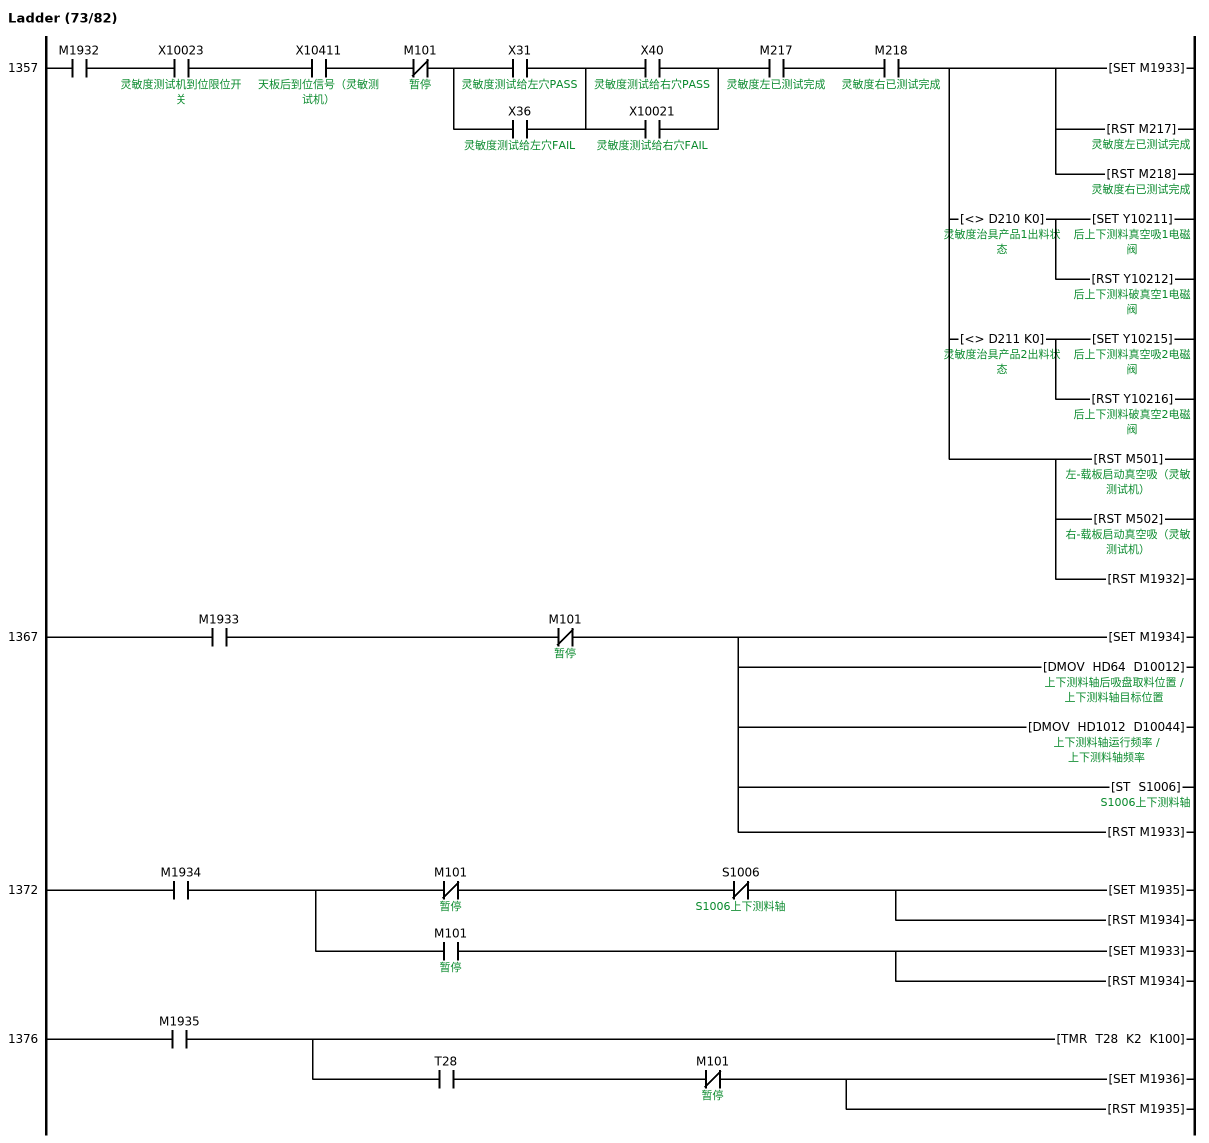
[picture p72: Ladder rows 1357-1376]
LD     M1932
AND    X10023	; 灵敏度测试机到位限位开关
AND    X10411	; 天板后到位信号（灵敏测试机）
ANI    M101	; 暂停
LD     X31	; 灵敏度测试给左穴PASS
OR     X36	; 灵敏度测试给左穴FAIL
ANB
LD     X40	; 灵敏度测试给右穴PASS
OR     X10021	; 灵敏度测试给右穴FAIL
ANB
AND    M217	; 灵敏度左已测试完成
AND    M218	; 灵敏度右已测试完成
SET    M1933
RST    M217	; 灵敏度左已测试完成
RST    M218	; 灵敏度右已测试完成
MPS
AND<>  D210 K0	; 灵敏度治具产品1出料状态
SET    Y10211	; 后上下测料真空吸1电磁阀
RST    Y10212	; 后上下测料破真空1电磁阀
MRD
AND<>  D211 K0	; 灵敏度治具产品2出料状态
SET    Y10215	; 后上下测料真空吸2电磁阀
RST    Y10216	; 后上下测料破真空2电磁阀
MPP
RST    M501	; 左-载板启动真空吸（灵敏测试机）
RST    M502	; 右-载板启动真空吸（灵敏测试机）
RST    M1932
LD     M1933
ANI    M101	; 暂停
SET    M1934
DMOV   HD64 D10012	; 上下测料轴后吸盘取料位置 / 上下测料轴目标位置
DMOV   HD1012 D10044	; 上下测料轴运行频率 / 上下测料轴频率
ST     S1006	; S1006上下测料轴
RST    M1933
LD     M1934
MPS
ANI    M101	; 暂停
ANI    S1006	; S1006上下测料轴
SET    M1935
RST    M1934
MPP
AND    M101	; 暂停
SET    M1933
RST    M1934
LD     M1935
TMR    T28 K2 K100
AND    T28
ANI    M101	; 暂停
SET    M1936
RST    M1935

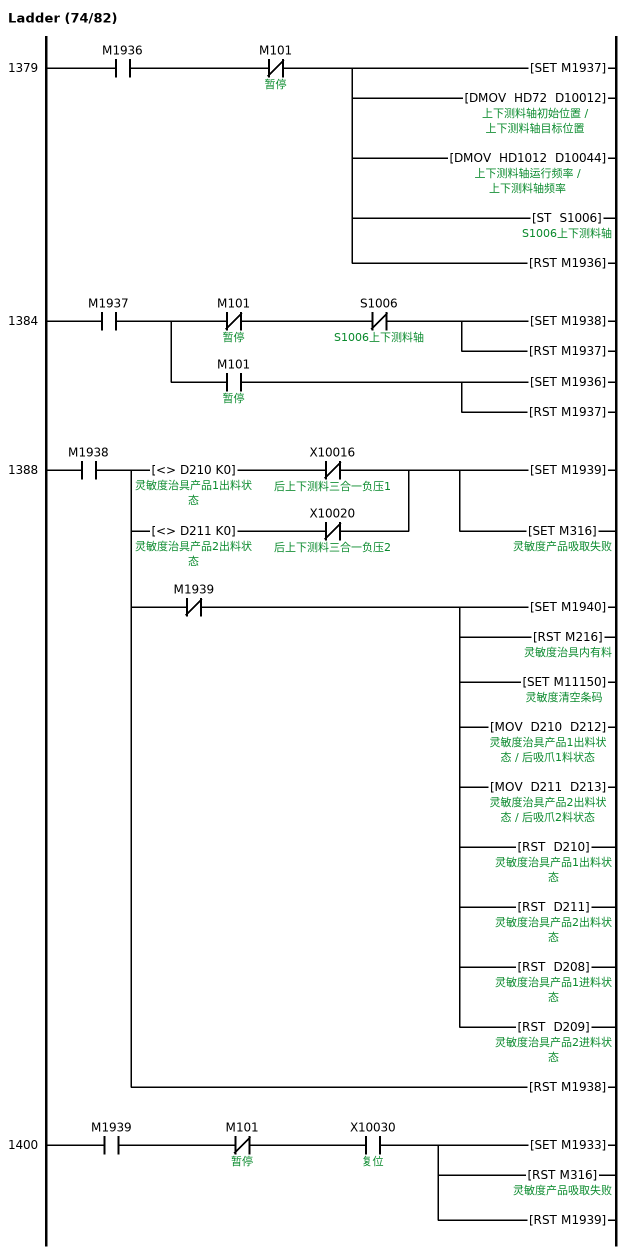
LD     M1936
ANI    M101	; 暂停
SET    M1937
DMOV   HD72 D10012	; 上下测料轴初始位置 / 上下测料轴目标位置
DMOV   HD1012 D10044	; 上下测料轴运行频率 / 上下测料轴频率
ST     S1006	; S1006上下测料轴
RST    M1936
LD     M1937
MPS
ANI    M101	; 暂停
ANI    S1006	; S1006上下测料轴
SET    M1938
RST    M1937
MPP
AND    M101	; 暂停
SET    M1936
RST    M1937
LD     M1938
MPS
LD<>   D210 K0	; 灵敏度治具产品1出料状态
ANI    X10016	; 后上下测料三合一负压1
LD<>   D211 K0	; 灵敏度治具产品2出料状态
ANI    X10020	; 后上下测料三合一负压2
ORB
ANB
SET    M1939
SET    M316	; 灵敏度产品吸取失败
MRD
ANI    M1939
SET    M1940
RST    M216	; 灵敏度治具内有料
SET    M11150	; 灵敏度清空条码
MOV    D210 D212	; 灵敏度治具产品1出料状态 / 后吸爪1料状态
MOV    D211 D213	; 灵敏度治具产品2出料状态 / 后吸爪2料状态
RST    D210	; 灵敏度治具产品1出料状态
RST    D211	; 灵敏度治具产品2出料状态
RST    D208	; 灵敏度治具产品1进料状态
RST    D209	; 灵敏度治具产品2进料状态
MPP
RST    M1938
LD     M1939
ANI    M101	; 暂停
AND    X10030	; 复位
SET    M1933
RST    M316	; 灵敏度产品吸取失败
RST    M1939

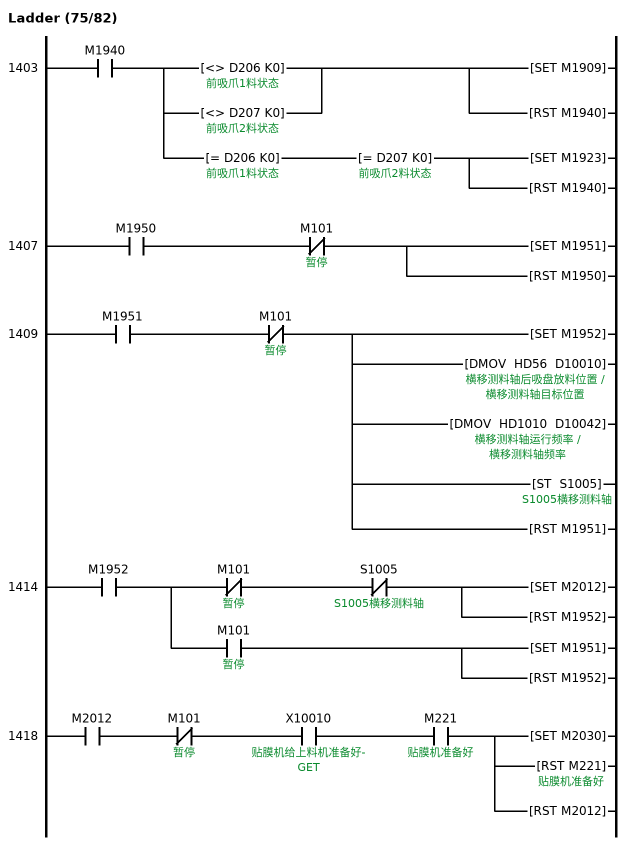
LD     M1940
MPS
LD<>   D206 K0	; 前吸爪1料状态
OR<>   D207 K0	; 前吸爪2料状态
ANB
SET    M1909
RST    M1940
MPP
AND=   D206 K0	; 前吸爪1料状态
AND=   D207 K0	; 前吸爪2料状态
SET    M1923
RST    M1940
LD     M1950
ANI    M101	; 暂停
SET    M1951
RST    M1950
LD     M1951
ANI    M101	; 暂停
SET    M1952
DMOV   HD56 D10010	; 横移测料轴后吸盘放料位置 / 横移测料轴目标位置
DMOV   HD1010 D10042	; 横移测料轴运行频率 / 横移测料轴频率
ST     S1005	; S1005横移测料轴
RST    M1951
LD     M1952
MPS
ANI    M101	; 暂停
ANI    S1005	; S1005横移测料轴
SET    M2012
RST    M1952
MPP
AND    M101	; 暂停
SET    M1951
RST    M1952
LD     M2012
ANI    M101	; 暂停
AND    X10010	; 贴膜机给上料机准备好-GET
AND    M221	; 贴膜机准备好
SET    M2030
RST    M221	; 贴膜机准备好
RST    M2012

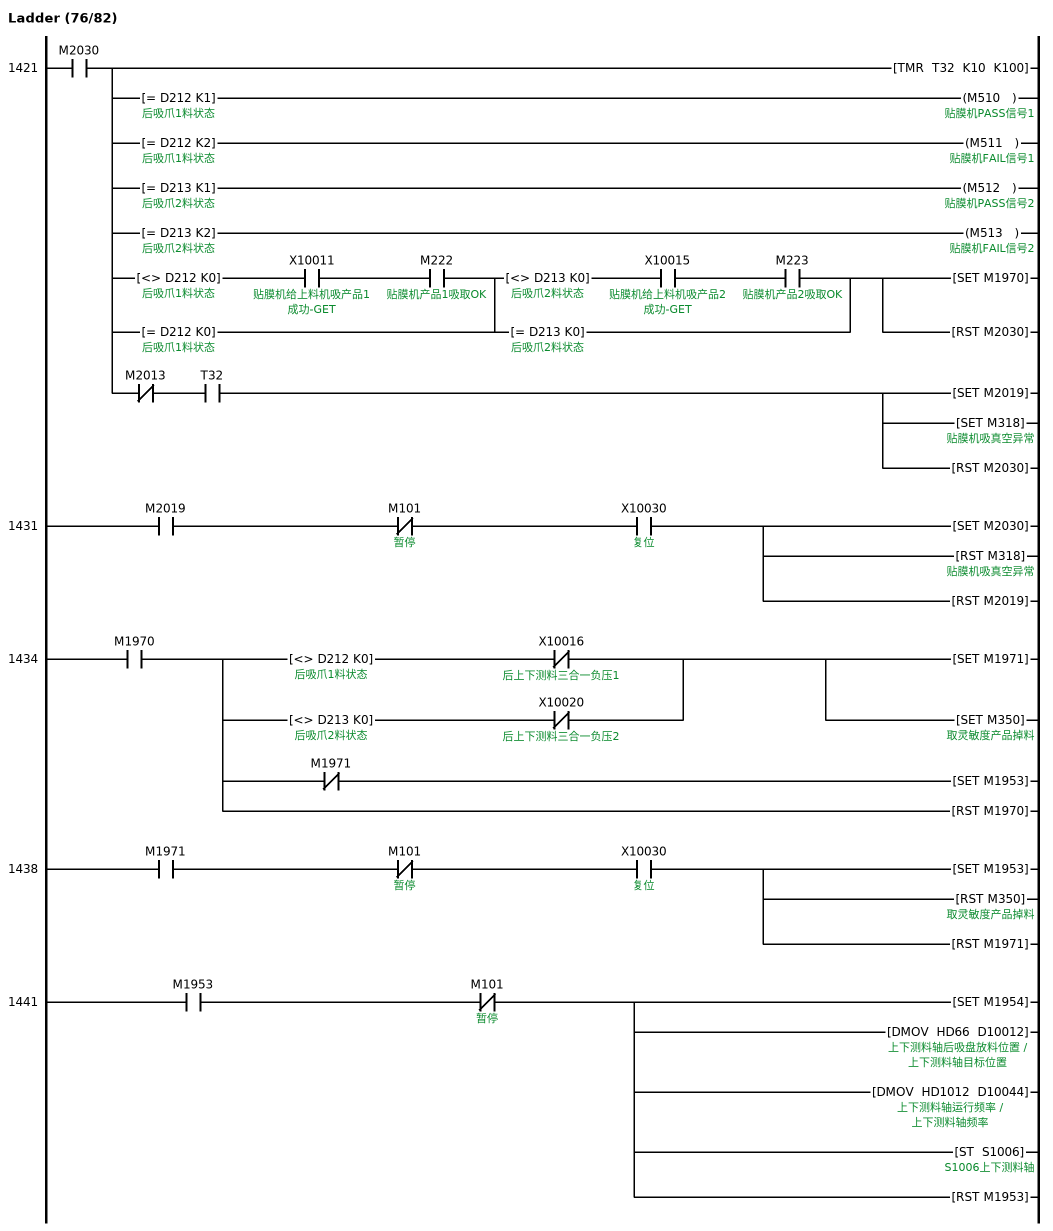
LD     M2030
TMR    T32 K10 K100
MPS
AND=   D212 K1	; 后吸爪1料状态
OUT    M510	; 贴膜机PASS信号1
MRD
AND=   D212 K2	; 后吸爪1料状态
OUT    M511	; 贴膜机FAIL信号1
MRD
AND=   D213 K1	; 后吸爪2料状态
OUT    M512	; 贴膜机PASS信号2
MRD
AND=   D213 K2	; 后吸爪2料状态
OUT    M513	; 贴膜机FAIL信号2
MRD
LD<>   D212 K0	; 后吸爪1料状态
AND    X10011	; 贴膜机给上料机吸产品1成功-GET
AND    M222	; 贴膜机产品1吸取OK
OR=    D212 K0	; 后吸爪1料状态
ANB
LD<>   D213 K0	; 后吸爪2料状态
AND    X10015	; 贴膜机给上料机吸产品2成功-GET
AND    M223	; 贴膜机产品2吸取OK
OR=    D213 K0	; 后吸爪2料状态
ANB
SET    M1970
RST    M2030
MPP
ANI    M2013
AND    T32
SET    M2019
SET    M318	; 贴膜机吸真空异常
RST    M2030
LD     M2019
ANI    M101	; 暂停
AND    X10030	; 复位
SET    M2030
RST    M318	; 贴膜机吸真空异常
RST    M2019
LD     M1970
MPS
LD<>   D212 K0	; 后吸爪1料状态
ANI    X10016	; 后上下测料三合一负压1
LD<>   D213 K0	; 后吸爪2料状态
ANI    X10020	; 后上下测料三合一负压2
ORB
ANB
SET    M1971
SET    M350	; 取灵敏度产品掉料
MRD
ANI    M1971
SET    M1953
MPP
RST    M1970
LD     M1971
ANI    M101	; 暂停
AND    X10030	; 复位
SET    M1953
RST    M350	; 取灵敏度产品掉料
RST    M1971
LD     M1953
ANI    M101	; 暂停
SET    M1954
DMOV   HD66 D10012	; 上下测料轴后吸盘放料位置 / 上下测料轴目标位置
DMOV   HD1012 D10044	; 上下测料轴运行频率 / 上下测料轴频率
ST     S1006	; S1006上下测料轴
RST    M1953

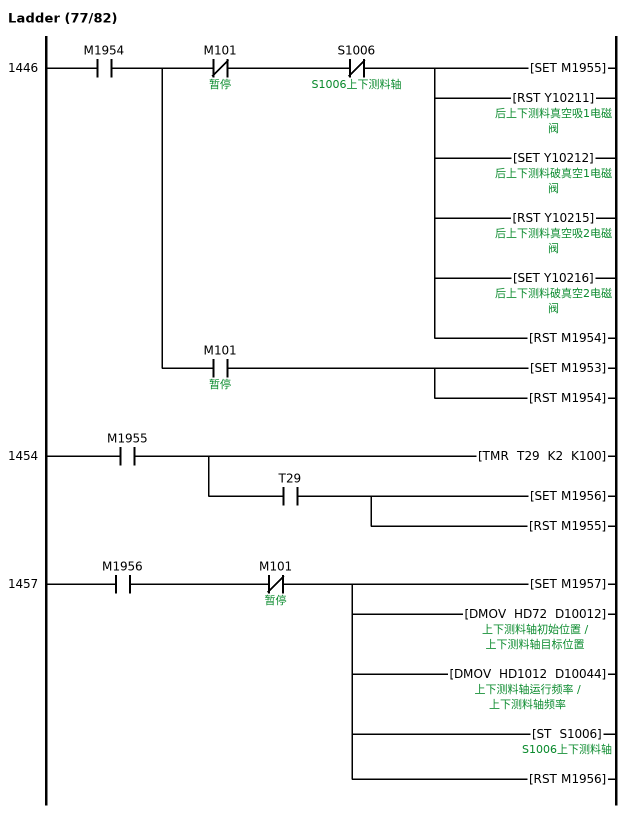
LD     M1954
MPS
ANI    M101	; 暂停
ANI    S1006	; S1006上下测料轴
SET    M1955
RST    Y10211	; 后上下测料真空吸1电磁阀
SET    Y10212	; 后上下测料破真空1电磁阀
RST    Y10215	; 后上下测料真空吸2电磁阀
SET    Y10216	; 后上下测料破真空2电磁阀
RST    M1954
MPP
AND    M101	; 暂停
SET    M1953
RST    M1954
LD     M1955
TMR    T29 K2 K100
AND    T29
SET    M1956
RST    M1955
LD     M1956
ANI    M101	; 暂停
SET    M1957
DMOV   HD72 D10012	; 上下测料轴初始位置 / 上下测料轴目标位置
DMOV   HD1012 D10044	; 上下测料轴运行频率 / 上下测料轴频率
ST     S1006	; S1006上下测料轴
RST    M1956

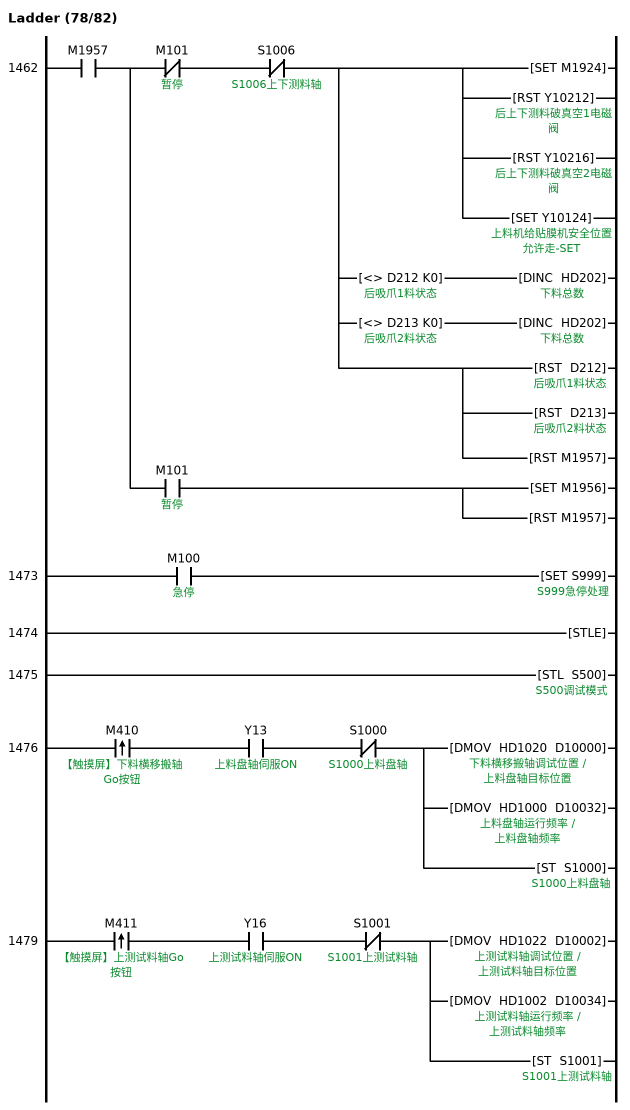
LD     M1957
MPS
ANI    M101	; 暂停
ANI    S1006	; S1006上下测料轴
SET    M1924
RST    Y10212	; 后上下测料破真空1电磁阀
RST    Y10216	; 后上下测料破真空2电磁阀
SET    Y10124	; 上料机给贴膜机安全位置允许走-SET
MPS
AND<>  D212 K0	; 后吸爪1料状态
DINC   HD202	; 下料总数
MRD
AND<>  D213 K0	; 后吸爪2料状态
DINC   HD202	; 下料总数
MPP
RST    D212	; 后吸爪1料状态
RST    D213	; 后吸爪2料状态
RST    M1957
MPP
AND    M101	; 暂停
SET    M1956
RST    M1957
LD     M100	; 急停
SET    S999	; S999急停处理
STLE
STL    S500	; S500调试模式
LDP    M410	; 【触摸屏】下料横移搬轴Go按钮
AND    Y13	; 上料盘轴伺服ON
ANI    S1000	; S1000上料盘轴
DMOV   HD1020 D10000	; 下料横移搬轴调试位置 / 上料盘轴目标位置
DMOV   HD1000 D10032	; 上料盘轴运行频率 / 上料盘轴频率
ST     S1000	; S1000上料盘轴
LDP    M411	; 【触摸屏】上测试料轴Go按钮
AND    Y16	; 上测试料轴伺服ON
ANI    S1001	; S1001上测试料轴
DMOV   HD1022 D10002	; 上测试料轴调试位置 / 上测试料轴目标位置
DMOV   HD1002 D10034	; 上测试料轴运行频率 / 上测试料轴频率
ST     S1001	; S1001上测试料轴

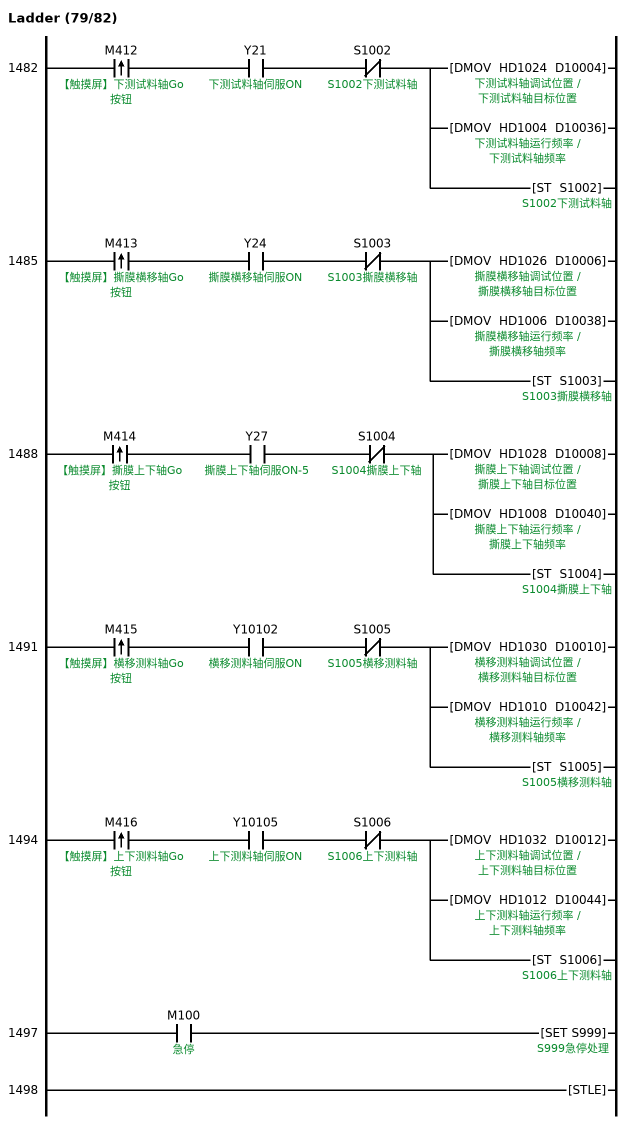
LDP    M412	; 【触摸屏】下测试料轴Go按钮
AND    Y21	; 下测试料轴伺服ON
ANI    S1002	; S1002下测试料轴
DMOV   HD1024 D10004	; 下测试料轴调试位置 / 下测试料轴目标位置
DMOV   HD1004 D10036	; 下测试料轴运行频率 / 下测试料轴频率
ST     S1002	; S1002下测试料轴
LDP    M413	; 【触摸屏】撕膜横移轴Go按钮
AND    Y24	; 撕膜横移轴伺服ON
ANI    S1003	; S1003撕膜横移轴
DMOV   HD1026 D10006	; 撕膜横移轴调试位置 / 撕膜横移轴目标位置
DMOV   HD1006 D10038	; 撕膜横移轴运行频率 / 撕膜横移轴频率
ST     S1003	; S1003撕膜横移轴
LDP    M414	; 【触摸屏】撕膜上下轴Go按钮
AND    Y27	; 撕膜上下轴伺服ON-5
ANI    S1004	; S1004撕膜上下轴
DMOV   HD1028 D10008	; 撕膜上下轴调试位置 / 撕膜上下轴目标位置
DMOV   HD1008 D10040	; 撕膜上下轴运行频率 / 撕膜上下轴频率
ST     S1004	; S1004撕膜上下轴
LDP    M415	; 【触摸屏】横移测料轴Go按钮
AND    Y10102	; 横移测料轴伺服ON
ANI    S1005	; S1005横移测料轴
DMOV   HD1030 D10010	; 横移测料轴调试位置 / 横移测料轴目标位置
DMOV   HD1010 D10042	; 横移测料轴运行频率 / 横移测料轴频率
ST     S1005	; S1005横移测料轴
LDP    M416	; 【触摸屏】上下测料轴Go按钮
AND    Y10105	; 上下测料轴伺服ON
ANI    S1006	; S1006上下测料轴
DMOV   HD1032 D10012	; 上下测料轴调试位置 / 上下测料轴目标位置
DMOV   HD1012 D10044	; 上下测料轴运行频率 / 上下测料轴频率
ST     S1006	; S1006上下测料轴
LD     M100	; 急停
SET    S999	; S999急停处理
STLE

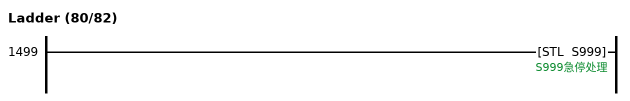
STL    S999	; S999急停处理

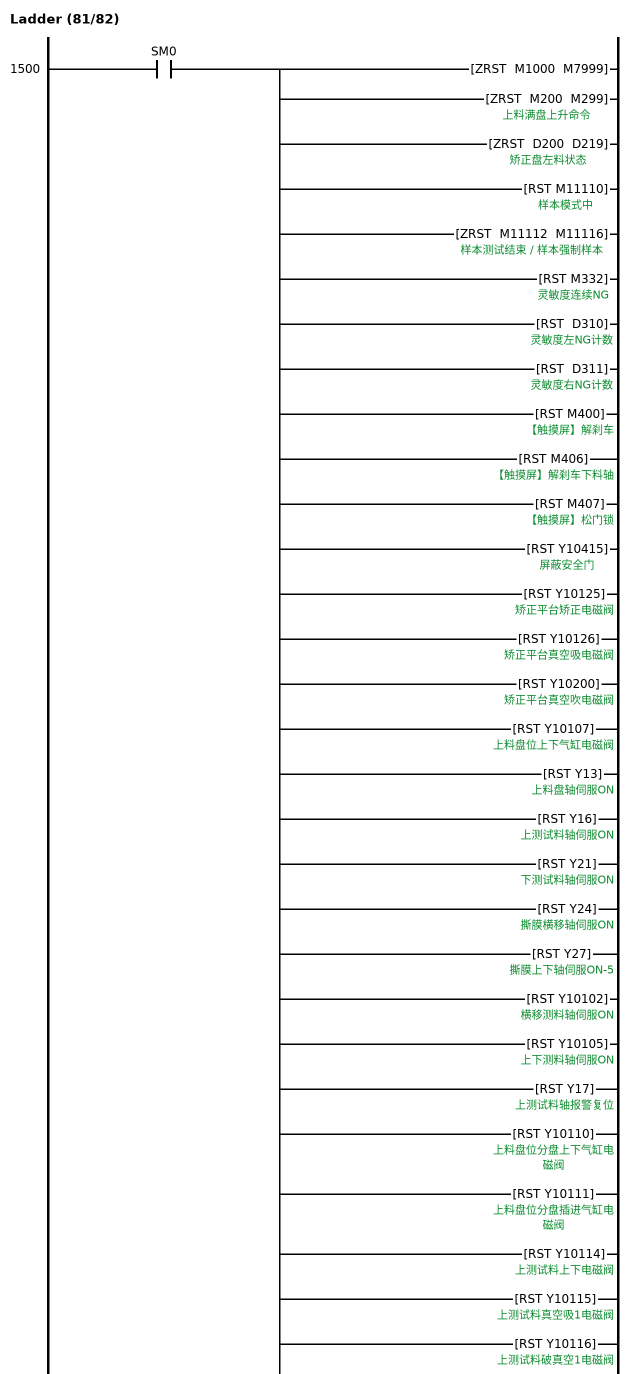
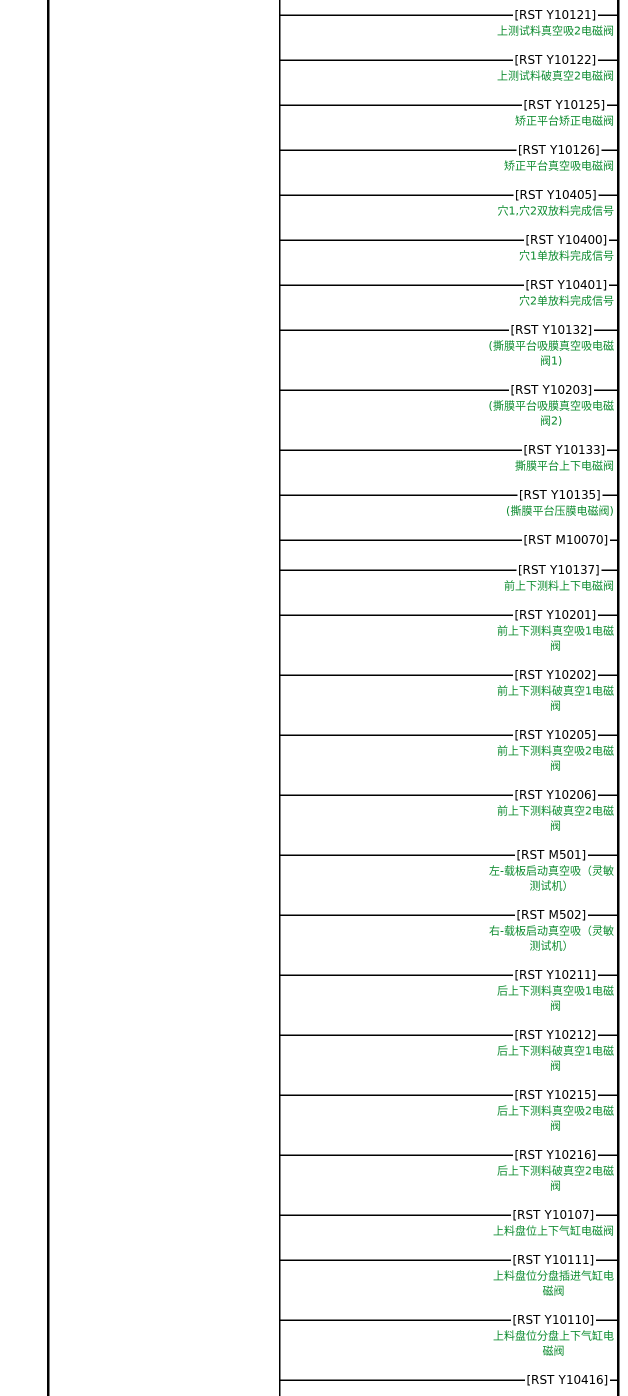
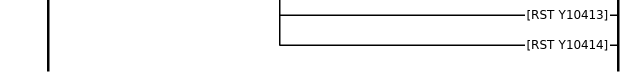
LD     SM0
ZRST   M1000 M7999
ZRST   M200 M299	; 上料满盘上升命令
ZRST   D200 D219	; 矫正盘左料状态
RST    M11110	; 样本模式中
ZRST   M11112 M11116	; 样本测试结束 / 样本强制样本
RST    M332	; 灵敏度连续NG
RST    D310	; 灵敏度左NG计数
RST    D311	; 灵敏度右NG计数
RST    M400	; 【触摸屏】解刹车
RST    M406	; 【触摸屏】解刹车下料轴
RST    M407	; 【触摸屏】松门锁
RST    Y10415	; 屏蔽安全门
RST    Y10125	; 矫正平台矫正电磁阀
RST    Y10126	; 矫正平台真空吸电磁阀
RST    Y10200	; 矫正平台真空吹电磁阀
RST    Y10107	; 上料盘位上下气缸电磁阀
RST    Y13	; 上料盘轴伺服ON
RST    Y16	; 上测试料轴伺服ON
RST    Y21	; 下测试料轴伺服ON
RST    Y24	; 撕膜横移轴伺服ON
RST    Y27	; 撕膜上下轴伺服ON-5
RST    Y10102	; 横移测料轴伺服ON
RST    Y10105	; 上下测料轴伺服ON
RST    Y17	; 上测试料轴报警复位
RST    Y10110	; 上料盘位分盘上下气缸电磁阀
RST    Y10111	; 上料盘位分盘插进气缸电磁阀
RST    Y10114	; 上测试料上下电磁阀
RST    Y10115	; 上测试料真空吸1电磁阀
RST    Y10116	; 上测试料破真空1电磁阀
RST    Y10121	; 上测试料真空吸2电磁阀
RST    Y10122	; 上测试料破真空2电磁阀
RST    Y10125	; 矫正平台矫正电磁阀
RST    Y10126	; 矫正平台真空吸电磁阀
RST    Y10405	; 穴1,穴2双放料完成信号
RST    Y10400	; 穴1单放料完成信号
RST    Y10401	; 穴2单放料完成信号
RST    Y10132	; (撕膜平台吸膜真空吸电磁阀1)
RST    Y10203	; (撕膜平台吸膜真空吸电磁阀2)
RST    Y10133	; 撕膜平台上下电磁阀
RST    Y10135	; (撕膜平台压膜电磁阀)
RST    M10070
RST    Y10137	; 前上下测料上下电磁阀
RST    Y10201	; 前上下测料真空吸1电磁阀
RST    Y10202	; 前上下测料破真空1电磁阀
RST    Y10205	; 前上下测料真空吸2电磁阀
RST    Y10206	; 前上下测料破真空2电磁阀
RST    M501	; 左-载板启动真空吸（灵敏测试机）
RST    M502	; 右-载板启动真空吸（灵敏测试机）
RST    Y10211	; 后上下测料真空吸1电磁阀
RST    Y10212	; 后上下测料破真空1电磁阀
RST    Y10215	; 后上下测料真空吸2电磁阀
RST    Y10216	; 后上下测料破真空2电磁阀
RST    Y10107	; 上料盘位上下气缸电磁阀
RST    Y10111	; 上料盘位分盘插进气缸电磁阀
RST    Y10110	; 上料盘位分盘上下气缸电磁阀
RST    Y10416
RST    Y10413
RST    Y10414

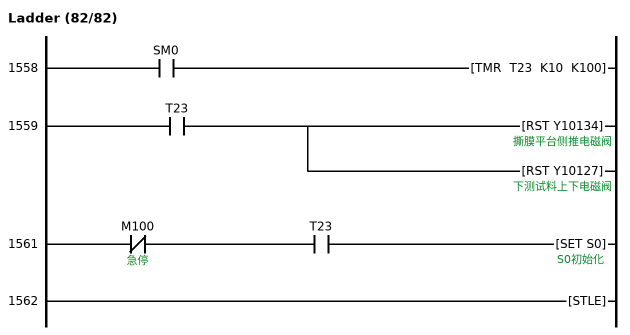
LD     SM0
TMR    T23 K10 K100
LD     T23
RST    Y10134	; 撕膜平台侧推电磁阀
RST    Y10127	; 下测试料上下电磁阀
LDI    M100	; 急停
AND    T23
SET    S0	; S0初始化
STLE

COMMENTS (devices not used above)
X0	上料盘轴差分板A
X1	上料盘轴差分板B
X3	上料轴光纤
X4	上料盘轴定位完成信号
X5	上料盘轴正转极限（远离电机）
X6	上料盘轴反转极限（靠近电机）
X7	上料盘轴原点
X16	分盘上下气缸SET传感器2
X17	分盘上下气缸RST传感器2
X21	光纤2-下空料盘满
X23	矫正负压信号2
X26	上测试料上下气缸SET传感器
X30	矫正气缸SET传感器
X32	矫正负压信号1
X35	收空盘光栅信号
X37	下测试料翻转气缸SET传感器
X41	撕膜平台吸左产品膜负压信号1
X10013	(撕膜平台吸右产品膜负压信号2)
X10034	排料完成【自机械手】
X10036	穴1样本取料
X10037	穴2样本取料
X10300	上测试轴取料光纤信号1
X10302	上测试轴取料光纤信号2
X10304	前测试轴取料光纤信号1
X10306	前测试轴取料光纤信号2
X10310	后测试轴取料光纤信号1
X10312	后测试轴取料光纤信号2
X10314	穴1样本PASS
X10315	穴1样本FAIL
X10316	穴2样本PASS
X10317	穴2样本FAIL
X10412	进入样本模式
Y10	脉冲口（备用）
Y11	脉冲口（备用）
Y14	卷胶带撕膜轴方向
Y22	下测试料轴报警复位
Y25	撕膜横移轴报警复位
Y10100	撕膜上下轴报警复位
Y10103	横移测料轴报警复位
Y10106	上下测料轴报警复位
Y10113	托盘夹紧气缸电磁阀
Y10130	下测试料压住电磁阀
Y10131	下测试料翻转电磁阀
Y10204	吸废膜真空吸电磁阀1
Y10207	吸废膜真空吸电磁阀2
Y10225	照明灯控制输出
Y10233	上料位反向信号 【至机械手】
Y10236	机械手可以取矫正盘【至机械手】
Y10403	上料机尾料信号
Y10404	样本取料完成信号
Y10406	联机复位信号
Y10407	上料机报警信号
Y10412	允许灵敏度开始测试信号（灵敏测试机）
M201	下空盘上升命令
M202	下空盘降格命令
M204	接空盘轴准备好
M219	接料平台空
M220	接料平台满
M307	下料上下搬轴指令未执行到位
M402	【触摸屏】上料盘电机升
M403	【触摸屏】上料盘电机降
M404	【触摸屏】下料盘电机升
M405	【触摸屏】下料盘电机降
M417	【触摸屏】下料上下搬轴Go按钮
M1030	空盘轴到底位
M1300	移载等待取盘
M10072	下料上下搬轴指令未执行到位
M10080	上盘步进轴正转
M10081	上盘步进轴反转
M10090	下盘步进轴正转
M10091	下盘步进轴反转
M11031	取下料区产品掉料
M20101	SCR-Running【机械手-运行】
M20103	SCR-Error【机械手-错误】
M20104	SCR-Estop【机械手-停止】
M20105	SCR-SafeguardOn【机械手-安全门】
M20106	SCR-SError【机械手-严重错误】
M20107	SCR-Warning【机械手-警告】
M20110	放料完成
S60	S60贴膜机下料机构
S99	S99急停处理
S1007	S1007下料上下搬运轴
D214	接料平台产品1状态
D215	接料平台产品2状态
D216	下料吸嘴产品1状态
D217	下料吸嘴产品2状态
D10014	下料上下搬轴目标位置
D10046	下料上下搬轴频率
HD160	下料横移搬运轴初始位置
HD162	下料横移搬运轴取料位置
HD164	下料横移搬运轴放料位置
HD170	下料上下搬运轴初始位置
HD172	下料上下搬运轴取料位置
HD174	下料上下搬运轴放料位置
HD208	UPH
HD1016	上盘步进轴运行频率
HD1018	下盘步进轴运行频率
HD1034	下料上下搬轴调试位置
HD2006	下料区产品吸取失败次数
HD2009	上测试料上下气缸报警次数
HD2010	前上下测料上下气缸报警次数
HD10000	下料横移搬轴运行频率
HD10002	上测试料轴运行频率
HD10004	下测试料轴运行频率
HD10006	撕膜横移轴运行频率
HD10008	撕膜上下轴运行频率
HD10010	横移测料轴运行频率
HD10012	上下测料轴运行频率
HD10014	下料上下搬轴运行频率
HD10016	上盘步进轴运行频率
HD10018	下盘步进轴运行频率